// TIA Portal V17 export
// export: Created 2025-03-05T08:03:37.7087517Z, ExportSetting WithDefaults, DisplayName Totally Integrated Automation Portal, DisplayVersion V17 Update 8, DisplayName TIA Portal Openness, DisplayVersion V17 Update 8, DisplayName TIA Portal Version Control Interface, DisplayVersion V17, DisplayName SINAMICS Startdrive Advanced, DisplayVersion V17 SP2, DisplayName SINAMICS Startdrive G110M, G120, G120C, G120D, G120P, G115D, DisplayVersion V17 SP2, DisplayName SINAMICS Startdrive G130, G150, S120, S150, SINAMICS MV, S210, DisplayVersion V17 SP2, DisplayName STEP 7 Professional, DisplayVersion V17 Update 8, DisplayName SINUMERIK ONE STEP 7 Toolbox, DisplayVersion V17 Update 12, DisplayName SINUMERIK 840D sl STEP 7 Toolbox, DisplayVersion V17 Update 12, DisplayName STEP 7 Safety, DisplayVersion V17 Update 6, DisplayName WinCC Advanced, DisplayVersion V17 Update 8
VAR_GLOBAL   // PLC tag table "TAGS_MARKS"
   Clock_Byte AT %MB1 : Byte;
   "M_0.1_SEC_10HZ" AT %M1.0 : Bool;   // 10HZ 0.1SEC
   "M_0.2_SEC_5Hz" AT %M1.1 : Bool;   // 5HZ 0.2SEC
   "M_0.4_SEC_2.5HZ" AT %M1.2 : Bool;   // 2.5HZ 0.4SEC
   "M_0.5_SEC_2HZ" AT %M1.3 : Bool;   // 2HZ 0.5SEC
   "M_0.8_SEC_1.25HZ" AT %M1.4 : Bool;   // 2.25HZ 0.8SEC
   "M_1.6_SEC_625HZ" AT %M1.6 : Bool;   // 0.625HZ 1.6SEC
   M_1_SEC_1HZ AT %M1.5 : Bool;   // 1HZ 1.0SEC
   "M_2_SEC_0.5HZ" AT %M1.7 : Bool;   // 0.5HZ 2.0SEC
   M_DUMMY_OFF AT %M0.3 : Bool;   // DUMMY OFF
   M_DUMMY_ON AT %M0.2 : Bool;   // DUMMY ON
   M_DUMMY_OUT AT %M0.4 : Bool;   // DUMMY OUT
   M_FIRST_SCAN AT %M0.6 : Bool;   // M FIRST SCAN
   M_NEW_START AT %M0.5 : Bool;   // NEW START / M NEW START
   M_ONE AT %M0.1 : Bool;   // ALWAYS ON
   M_REVISAR_FALTA_ALGO AT %M2.3 : Bool;   // REVISAR FALTA ALGO DE PROGRAMACIÓN
   M_TEMPORARY_USE_OEM AT %M5.0 : Bool;   // M_TEMPORARY_USE_OEM(CONFIGURE CORRECTLY AND DELETE) / M FOR TEMPORARY USE (OEM)
   M_ZERO AT %M0.0 : Bool;   // ALWAYS OFF
   NETWORK_CHECK AT %M0.7 : Bool;   // ADAPT NETWORK LOGIC ACCORDING TO MACHINE STRUCTURE
   Softkey_Input_Byte AT %IB124 : Byte;
END_VAR
